Fanuc KAREL source: kb00066.KL

-- PROVISIONAL review KL for V1013-1; original PC SHA256 9d8e6f1148202f2c84f5c358e54dcb9f78e1256580a9e0eeb024f4a0fbfdd796
-- Incomplete behavior may be omitted. Consult companion uncertainty JSON. Do not deploy.
PROGRAM KB00066
%NOLOCKGROUP
BEGIN
  -- UNRESOLVED_PC offsets 5-14; opcodes 3F,75
  -- UNRESOLVED_PC offsets 19-26; opcodes 9D,23
  -- UNRESOLVED_PC offsets 31-38; opcodes 9D,23
  -- UNRESOLVED_PC offsets 43-50; opcodes 9D,23
  -- UNRESOLVED_PC offsets 55-62; opcodes 9D,23
  -- UNRESOLVED_PC offsets 67-74; opcodes 9D,23
  -- UNRESOLVED_PC offsets 79-139; opcodes 27,22,2A,22,22,22,22,22,22,22,22,31
  -- UNRESOLVED_PC offsets 144-148; opcodes 7F
END KB00066
